Yaskawa INFORM job: ramp_07_08_23_planes_program.JBI

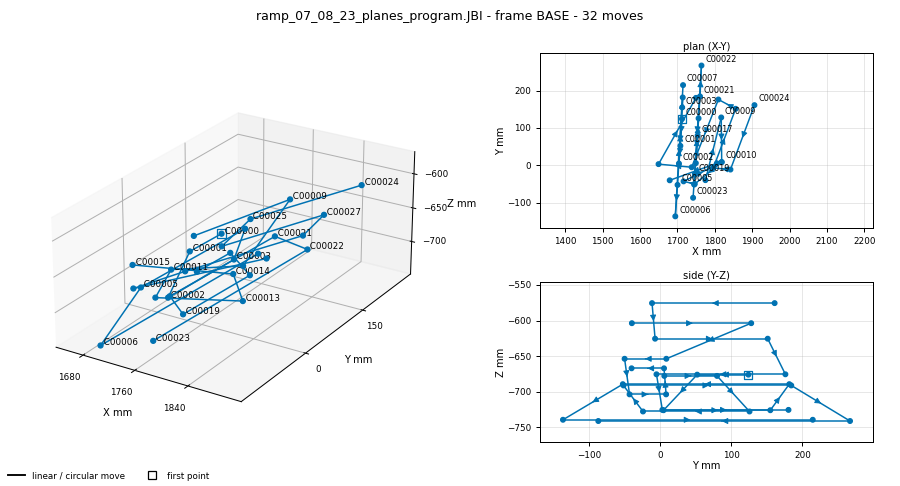
[picture p0: tool path of ramp_07_08_23_planes_program.JBI in frame BASE, 32 of 38 moves have a stored position in this frame; points joined in program order, loops and branches not executed]
/JOB
//NAME ramp_07_08_23_planes_program
//POS
///NPOS 32,0,32,0,0,0
///TOOL 0
///POSTYPE BASE
///RECTAN
///RCONF 0,0,0,0,0,0,0,0,0,0,0,0,0,0,0,0,0,0,0,0,0,0,0,0
C00000=1712.202900,124.152125,-676.042305,175.000000,-88.995474,-5.000000
C00001=1707.892900,52.198325,-676.042305,175.000000,-88.995474,-5.000000
C00002=1703.982900,4.925425,-726.042305,175.000000,-88.995474,-5.000000
C00003=1712.692900,154.936125,-726.042305,175.000000,-88.995474,-5.000000
C00004=1714.142900,181.593825,-689.439765,180.000000,-60.000000,0.000000
C00005=1700.282900,-52.287575,-689.439765,180.000000,-60.000000,0.000000
C00006=1694.272900,-136.395575,-739.439765,180.000000,-60.000000,0.000000
C00007=1715.002900,214.578425,-739.439765,180.000000,-60.000000,0.000000
C00008=1774.846050,-39.562785,-603.737900,175.000000,-59.649120,-5.000000
C00009=1817.121050,128.097215,-603.737900,175.000000,-59.649120,-5.000000
C00010=1818.396550,8.837215,-653.737900,175.000000,-59.649120,-5.000000
C00011=1746.348750,-49.802785,-653.737900,175.000000,-59.649120,-5.000000
C00012=1716.375050,-42.842785,-703.737900,175.000000,-59.649120,-5.000000
C00013=1818.269050,8.527215,-703.737900,175.000000,-59.649120,-5.000000
C00014=1805.446110,5.587215,-667.135360,180.000000,-60.000000,0.000000
C00015=1679.306150,-40.002785,-667.135360,180.000000,-60.000000,0.000000
C00016=1749.200900,5.984735,-677.796721,175.000000,-89.572480,-5.000000
C00017=1753.980900,80.064915,-677.796721,175.000000,-89.572480,-5.000000
C00018=1756.500900,125.724515,-727.796721,175.000000,-89.572480,-5.000000
C00019=1746.690900,-23.926585,-727.796721,175.000000,-89.572480,-5.000000
C00020=1744.770900,-51.387385,-691.194181,180.000000,-60.000000,0.000000
C00021=1760.340900,184.380515,-691.194181,180.000000,-60.000000,0.000000
C00022=1764.260900,266.960515,-741.194181,180.000000,-60.000000,0.000000
C00023=1741.900900,-86.732985,-741.194181,180.000000,-60.000000,0.000000
C00024=1905.970550,161.005900,-575.546150,175.000000,-46.004717,-5.000000
C00025=1841.798050,-11.234100,-575.546150,175.000000,-46.004717,-5.000000
C00026=1795.956050,-6.954100,-625.546150,175.000000,-46.004717,-5.000000
C00027=1855.748850,151.275900,-625.546150,175.000000,-46.004717,-5.000000
C00028=1809.502050,176.135900,-675.546150,175.000000,-46.004717,-5.000000
C00029=1738.125050,-5.014100,-675.546150,175.000000,-46.004717,-5.000000
C00030=1649.465050,3.245900,-725.546150,175.000000,-46.004717,-5.000000
C00031=1749.467050,180.485900,-725.546150,175.000000,-46.004717,-5.000000
///POSTYPE PULSE
///PULSE
EC00000=0
EC00001=0
EC00002=0
EC00003=0
EC00004=0
EC00005=0
EC00006=0
EC00007=0
EC00008=92160
EC00009=92160
EC00010=92160
EC00011=92160
EC00012=92160
EC00013=92160
EC00014=92160
EC00015=92160
EC00016=184320
EC00017=184320
EC00018=184320
EC00019=184320
EC00020=184320
EC00021=184320
EC00022=184320
EC00023=184320
EC00024=276480
EC00025=276480
EC00026=276480
EC00027=276480
EC00028=276480
EC00029=276480
EC00030=276480
EC00031=276480
//INST
///DATE 2023/08/07 12:29
///ATTR SC,RW,RJ
////FRAME BASE
///GROUP1 RB1,ST1
NOP
MOVJ P009 EX000 VJ=15.00
MOVJ P009 VJ=15.00
MOVJ C00000 EC00000 VJ=15.0
CALL JOB:SPYON
MOVL C00001 EC00001 V=150.0
MOVL C00002 EC00002 V=150.0
MOVL C00003 EC00003 V=150.0
MOVL C00004 EC00004 V=150.0
MOVL C00005 EC00005 V=150.0
MOVL C00006 EC00006 V=150.0
MOVL C00007 EC00007 V=150.0
CALL JOB:SPYOF
MOVJ P009 VJ=15.00
MOVJ C00008 EC00008 VJ=15.0
CALL JOB:SPYON
MOVL C00009 EC00009 V=150.0
MOVL C00010 EC00010 V=150.0
MOVL C00011 EC00011 V=150.0
MOVL C00012 EC00012 V=150.0
MOVL C00013 EC00013 V=150.0
MOVL C00014 EC00014 V=150.0
MOVL C00015 EC00015 V=150.0
CALL JOB:SPYOF
MOVJ P009 VJ=15.00
MOVJ C00016 EC00016 VJ=15.0
CALL JOB:SPYON
MOVL C00017 EC00017 V=150.0
MOVL C00018 EC00018 V=150.0
MOVL C00019 EC00019 V=150.0
MOVL C00020 EC00020 V=150.0
MOVL C00021 EC00021 V=150.0
MOVL C00022 EC00022 V=150.0
MOVL C00023 EC00023 V=150.0
CALL JOB:SPYOF
MOVJ P009 VJ=15.00
MOVJ C00024 EC00024 VJ=15.0
CALL JOB:SPYON
MOVL C00025 EC00025 V=150.0
MOVL C00026 EC00026 V=150.0
MOVL C00027 EC00027 V=150.0
MOVL C00028 EC00028 V=150.0
MOVL C00029 EC00029 V=150.0
MOVL C00030 EC00030 V=150.0
MOVL C00031 EC00031 V=150.0
CALL JOB:SPYOF
MOVJ P009 VJ=15.00
END
